TYPE ST_PTM :
STRUCT
(* General PTM Structure
Each PTM might have a serial control structure, but all will have a general supervisory control structure

NOTE: This is an archetype, use an extension of this structure for a specific pump (or make one).

*)

(* Controls *)
	{attribute 'pytmc' := '
	pv: RUN_SW;
	io: io;
	'}
	xRunSW	:	BOOL;
	{attribute 'pytmc' := '
	pv: RST_SW;
	io: io;
	'}
	xResetSW	:	BOOL; //For resetting faults
	{attribute 'pytmc' := '
    pv: RUN_DO;
	io: i;
	'}
	q_RunDO 	:	BOOL;

(* Readbacks *)
    {attribute 'pytmc' := '
	pv: ILK_OK;
	field: ZNAM ILK ACTIVE;
	field: ONAM ILK OK;
	io: i;
	'}
	xExtRunOk	:	BOOL; (* also a control *)
	{attribute 'pytmc' := '
    pv: ACCEL;
	io: i;
	'}
	i_xAccel	:	BOOL;
	{attribute 'pytmc' := '
    pv: AT_SPD;
	io: i;
	'}
	i_xAtSpd	:	BOOL;
	{attribute 'pytmc' := '
	pv: SPEED_RDBK;
	io: i;
	'}
	i_diCurSpd	:	DINT;
	
	xCommTimeout	:	BOOL := TRUE;  (* Initialized true since we haven't talked to pump yet *)
(* Alarm Outputs *)
	{attribute 'pytmc' := '
    pv: FAULT;
	io: i;
	'}
	i_xFault		:	BOOL; (*FAULT*)
	{attribute 'pytmc' := '
    pv: WARN;
	io: i;
	'}
	i_xWarn		:	BOOL; (* warning *)
	{attribute 'pytmc' := '
    pv: ALARM;
	io: i;
	'}
	i_xALARM	:	BOOL; (* ALARM *)
	
(* IWS instructions *)
	xActive	:	BOOL; // this bit is set to add the pump to the system
	iPumpGrp 	:	INT; // all members of a pump group start at the same time
	
(* Operational Setpoints *)
	rForelineSP	:	REAL := 0.5;
	
	{attribute 'pytmc' := '
    pv: BackingPressureSP;
	io: io;
	'}
	rBackingPressureSP : REAL := 0.01;
	{attribute 'pytmc' := '
    pv: InletPressureSP;
	io: io;
	'}
	rInletPressureSP : REAL := 0.5;
(*State*)	
	{attribute 'pytmc' := '
	pv: STATE;
	field: ZRST STOPPED;
	field: ONST STARTING;
	field: TWST RUNNING;
	field: THST FAULT;
	io: i;
	'}

	eState	:	E_PumpState;
	
	{attribute 'pytmc' := '
	pv: Current_MON;
	io: i;
	'}
	i_iCurrentMon : INT; // Voltage to the output current of motor 0->5V 0->10A


END_STRUCT
END_TYPE

(* stored: Version 1.1.0.1, ProductVersion 3.1.4024.0
   DUT ST_PTM: Id {4cff5a41-fc78-4938-9468-a980c788ccb5} *)
